(* Logix 5000 project; controller CPU_01 1756-L85E rev 36.11; software revision 36.00 *)
// CODE TESTING 20250421

TASK MainTask (continuous, watchdog 500 ms) : MainProgram, AlarmManagement, DesignPatters

MODULES
   Local : 1756-L85E (ICP 2, rev 36.11)
      INPUTS : vendor 1 type 0 code 15 (ICP 3, rev 1.1, Output RPI 50 ms)
      OUTPUT : vendor 1 type 0 code 15 (ICP 4, rev 1.1, Output RPI 50 ms)
END_MODULES

TYPE IBN_Programming :
STRUCT
   DEBUG : BOOL;   // DEBUGGING
   TODO : BOOL;   // TODO
   BYPASS : BOOL;   // BYPASS - DONOT REMOVE
   ALWAYS_OFF : BOOL;   // ALWAY OFF
   ALWAYS_ON : BOOL;   // ALWAY ON
   OUTPUTS : DINT[25];   // TEST BIT OUTPUTS
   SERIAL_NUMBER : DINT[25];   // OPEN ISSUES
END_STRUCT
END_TYPE

TYPE UDT_FiveStepMethod :
STRUCT
   TriggerPrecodition : BOOL;
   Safe : BOOL;
   Command : BOOL;
   InPosition : BOOL;
   TimeOutFault : BOOL;
END_STRUCT
END_TYPE

TYPE UDT_Missions :
STRUCT
   Missions : DINT;
   Start : DINT;
   Done : DINT;
END_STRUCT
END_TYPE

ADD_ON_INSTRUCTION AO_HANDLE_COMMAND_PANEL_BUTTONS_HARDWARE   (* revision 1.0 *)

ROUTINE Logic   (* structured text *)
   
END_ROUTINE
END_ADD_ON_INSTRUCTION

ADD_ON_INSTRUCTION AOI_Flasher   (* revision 1.0 *)
VAR_OUTPUT
   Output : BOOL; {access None, required}
END_VAR
VAR_INPUT
   TimerPreset_2 : DINT; {access None, required}
   TimerPreset_1 : DINT; {access None, required}
END_VAR
VAR
   Timer : TIMER[2]; {access None}
END_VAR

ROUTINE Logic   (* ladder *)
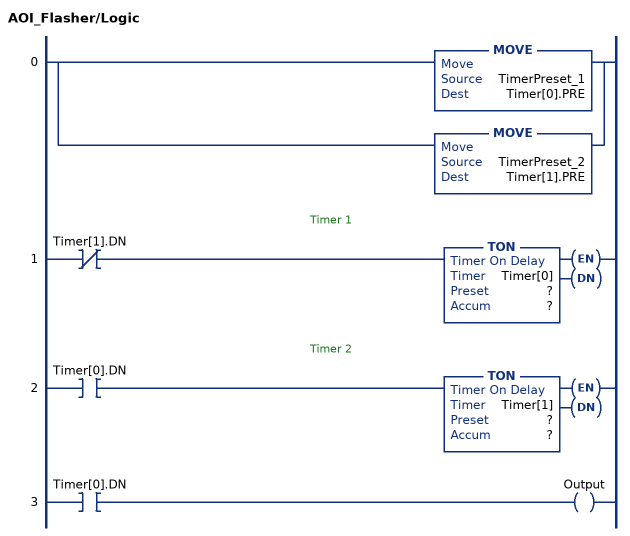
   0: [MOVE(TimerPreset_1,Timer[0].PRE) ,MOVE(TimerPreset_2,Timer[1].PRE) ];
   // Timer 1
   1: XIO(Timer[1].DN)TON(Timer[0],?,?);
   // Timer 2
   2: XIC(Timer[0].DN)TON(Timer[1],?,?);
   3: XIC(Timer[0].DN)OTE(Output);
END_ROUTINE
END_ADD_ON_INSTRUCTION

ADD_ON_INSTRUCTION AOI_Flasher_01   (* revision 1.0 *)
VAR_OUTPUT
   FLASHER_500ms_Led : BOOL; {access Read Only, required}
END_VAR
VAR
   FLASHER_500ms : FBD_TIMER; {access None}
END_VAR

ROUTINE Logic   (* structured text *)
   (* Declare Timer and Tag Variables *)
   IF NOT FLASHER_500ms.DN THEN
   	FLASHER_500ms.PRE := 1000;
   	FLASHER_500ms.EN := 1;
   	tonr(FLASHER_500ms);
   
   END_IF;
   
   IF FLASHER_500ms.ACC >= 1000 THEN
       FLASHER_500ms_Led := 1;
   ELSE
       FLASHER_500ms_Led := 0;
   END_IF;
   
   
END_ROUTINE
END_ADD_ON_INSTRUCTION

VAR_GLOBAL   (* controller tags *)
   DateTimeFromPLC : DINT[7] := ([0] := 2025, [1] := 4, [2] := 21, [3] := 16, [4] := 49, [5] := 42, [6] := 773920);
        [0]   // Year
        [1]   // Month
        [2]   // Day
        [3]   // Hours
        [4]   // Minute
        [5]   // Seconds
        [6]   // Microseconds
   IBN_DHF : IBN_Programming := (ALWAYS_ON := 1, SERIAL_NUMBER[1] := 24);
        .SERIAL_NUMBER[0].0   // 001: Timer not working
        .OUTPUTS[0].0   // 000: Spare
        .OUTPUTS[0].1   // 001: Basic Flasher bit
        .SERIAL_NUMBER[0].1   // 002: Create a trigger for getting the time
   R6 : CONTROL[25] := ([3].LEN := 4, [3].POS := 3);
   SterileWaterRinse_Array : DINT[2,20] := ([0,0] := 1, [0,1] := 2, [0,2] := 4, [0,3] := 12);
   SterileWaterRinse_Bits : DINT[8] := ([0] := 12, [2] := 7);
END_VAR

PROGRAM AlarmManagement   (* main routine R000_MainRouting *)
VAR
   AlarmMessage : BOOL[64] := ([0] := 1, [2] := 1);
        [0]   // 1000: Motor overload tripped
        [1]   // 1001: Pump over tempature
   AlarmTimers : TIMER[16] := ([0].PRE := 5000, [0].ACC := 5000, [0].EN := 1, [0].DN := 1);
   AlarmTrigger : BOOL[64];
   Messages : BOOL[64];
   MotorOverLoad : BOOL;
   MotorStart : BOOL := 1;
   PumpTemperature : DINT;
END_VAR

ROUTINE R000_MainRouting   (* structured text *)
   // Blocks
   jsr(R020_AlarmManagement);
   
END_ROUTINE

ROUTINE R020_AlarmManagement   (* ladder *)
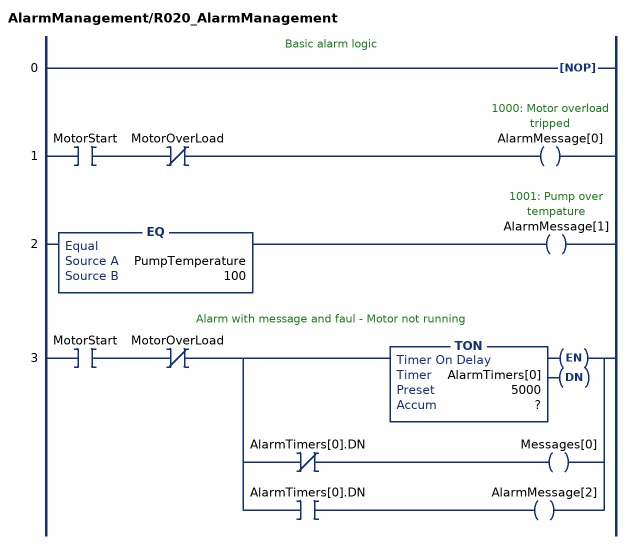
   // Basic alarm logic
   0: NOP();
   1: XIC(MotorStart)XIO(MotorOverLoad)OTE(AlarmMessage[0]);
   2: EQ(PumpTemperature,100)OTE(AlarmMessage[1]);
   // Alarm with message and faul - Motor not running
   3: XIC(MotorStart)XIO(MotorOverLoad)[TON(AlarmTimers[0],?,?) ,XIO(AlarmTimers[0].DN) OTE(Messages[0]) ,XIC(AlarmTimers[0].DN) OTE(AlarmMessage[2]) ];
END_ROUTINE
END_PROGRAM

PROGRAM DesignPatters   (* main routine R000_MainRoutine *)
VAR
   AutoMode : BOOL;
   AutoModePB : BOOL;
   Command : BOOL;
   EStopOK : BOOL;
   FaultTimeOut : BOOL;
   FaultTimer : TIMER := (PRE := 1000);
   FaultTimerReset : BOOL;
   Flasher1 : BOOL;
   Flasher_10 : AOI_Flasher_01;
   Flasher_1_sec : BOOL;
   Flasher_5000hz : AOI_Flasher := (TimerPreset_2 := 500, TimerPreset_1 := 500);
   FromSeqLogic : BOOL;
   InPosition : BOOL;
   LED : BOOL;
   LED_2 : BOOL;
   ManualMode : BOOL := 1;
   ManualModePB : BOOL;
   MissionsDone : DINT;   // Mssions complete
        .1   // Mission 1 done
   MissionsStart : DINT;   // Mssions complete
        .1   // Mission 1 done
   Mode : DINT := 1;
   ModePB : DINT := 1;
   PushButton : BOOL;
   Safe : BOOL;
   Sensor : BOOL;
   TimeOutFault : BOOL;
   TON_Flasher_1_sec : TIMER := (PRE := 2000, ACC := 147, EN := 1, TT := 1);
   TriggerPrecondition : BOOL;
   ValveMissions : UDT_Missions := (Missions := 1);
        .Missions.0   // No mission
        .Missions.1   // Mission 1
        .Missions.2   // Mission 2
END_VAR

ROUTINE R000_MainRoutine   (* ladder *)
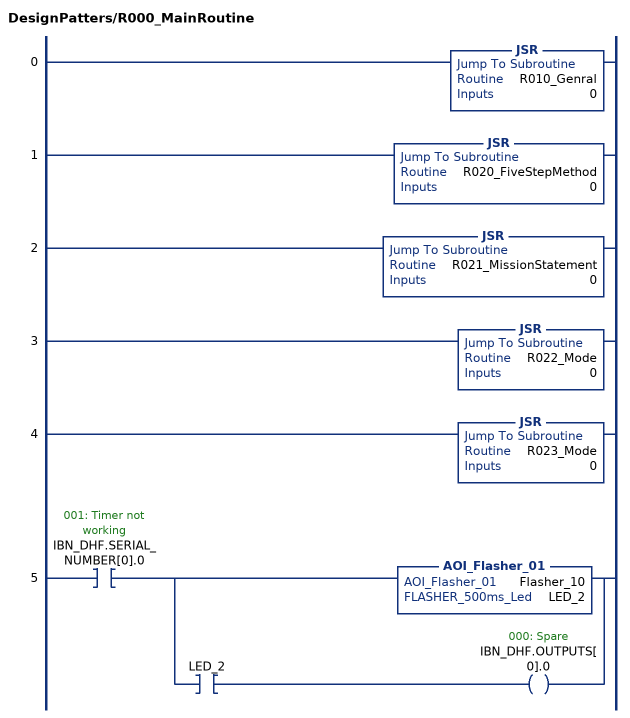
   0: JSR(R010_Genral,0);
   1: JSR(R020_FiveStepMethod,0);
   2: JSR(R021_MissionStatement,0);
   3: JSR(R022_Mode,0);
   4: JSR(R023_Mode,0);
   5: XIC(IBN_DHF.SERIAL_NUMBER[0].0)[AOI_Flasher_01(Flasher_10,LED_2) ,XIC(LED_2) OTE(IBN_DHF.OUTPUTS[0].0) ];
END_ROUTINE

ROUTINE R010_Genral   (* ladder *)
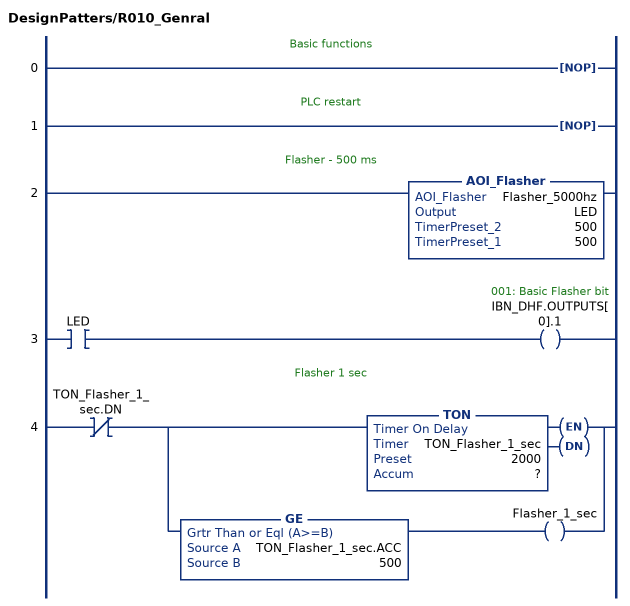
   // Basic functions
   0: NOP();
   // PLC restart
   1: NOP();
   // Flasher - 500 ms
   2: AOI_Flasher(Flasher_5000hz,LED,500,500);
   3: XIC(LED)OTE(IBN_DHF.OUTPUTS[0].1);
   // Flasher 1 sec
   4: XIO(TON_Flasher_1_sec.DN)[TON(TON_Flasher_1_sec,?,?) ,GE(TON_Flasher_1_sec.ACC,500) OTE(Flasher_1_sec) ];
END_ROUTINE

ROUTINE R020_FiveStepMethod   (* ladder *)
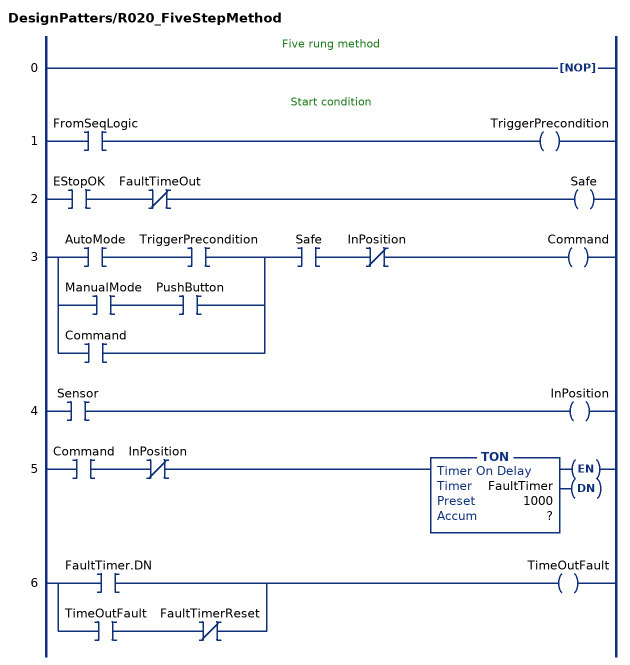
   // Five rung method
   0: NOP();
   // Start condition
   1: XIC(FromSeqLogic)OTE(TriggerPrecondition);
   2: XIC(EStopOK)XIO(FaultTimeOut)OTE(Safe);
   3: [XIC(AutoMode) XIC(TriggerPrecondition) ,XIC(ManualMode) XIC(PushButton) ,XIC(Command) ]XIC(Safe)XIO(InPosition)OTE(Command);
   4: XIC(Sensor)OTE(InPosition);
   5: XIC(Command)XIO(InPosition)TON(FaultTimer,?,?);
   6: [XIC(FaultTimer.DN) ,XIC(TimeOutFault) XIO(FaultTimerReset) ]OTE(TimeOutFault);
END_ROUTINE

ROUTINE R021_MissionStatement   (* ladder *)
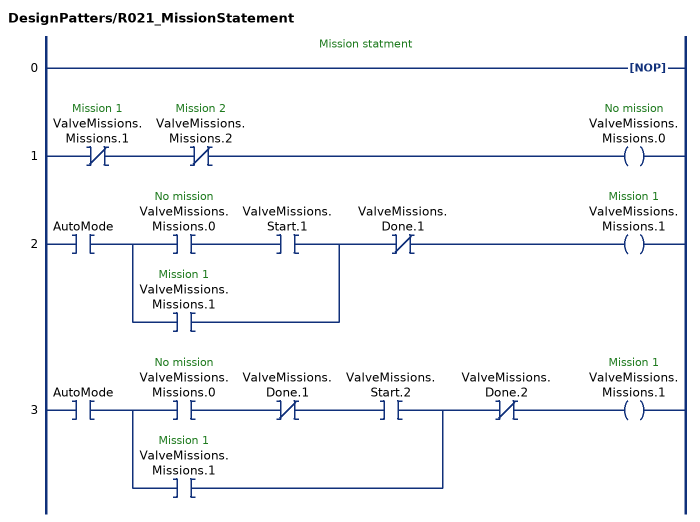
   // Mission statment
   0: NOP();
   1: XIO(ValveMissions.Missions.1)XIO(ValveMissions.Missions.2)OTE(ValveMissions.Missions.0);
   2: XIC(AutoMode)[XIC(ValveMissions.Missions.0) XIC(ValveMissions.Start.1) ,XIC(ValveMissions.Missions.1) ]XIO(ValveMissions.Done.1)OTE(ValveMissions.Missions.1);
   3: XIC(AutoMode)[XIC(ValveMissions.Missions.0) XIO(ValveMissions.Done.1) XIC(ValveMissions.Start.2) ,XIC(ValveMissions.Missions.1) ]XIO(ValveMissions.Done.2)OTE(ValveMissions.Missions.1);
END_ROUTINE

ROUTINE R022_Mode   (* ladder *)
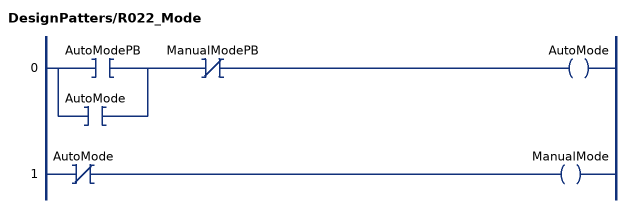
   0: [XIC(AutoModePB) ,XIC(AutoMode) ]XIO(ManualModePB)OTE(AutoMode);
   1: XIO(AutoMode)OTE(ManualMode);
END_ROUTINE

ROUTINE R023_Mode   (* ladder *)
// Three mode selection
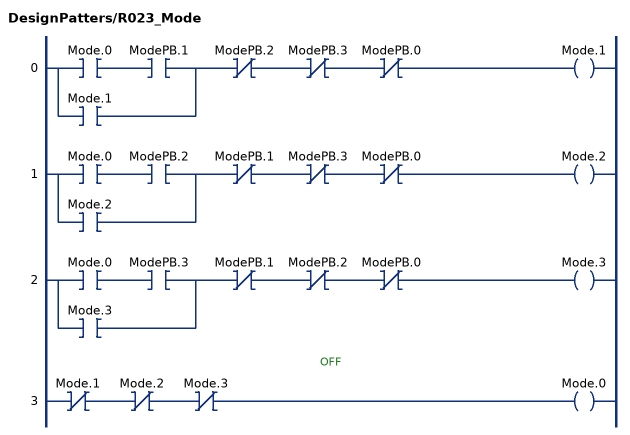
   0: [XIC(Mode.0) XIC(ModePB.1) ,XIC(Mode.1) ]XIO(ModePB.2)XIO(ModePB.3)XIO(ModePB.0)OTE(Mode.1);
   1: [XIC(Mode.0) XIC(ModePB.2) ,XIC(Mode.2) ]XIO(ModePB.1)XIO(ModePB.3)XIO(ModePB.0)OTE(Mode.2);
   2: [XIC(Mode.0) XIC(ModePB.3) ,XIC(Mode.3) ]XIO(ModePB.1)XIO(ModePB.2)XIO(ModePB.0)OTE(Mode.3);
   // OFF
   3: XIO(Mode.1)XIO(Mode.2)XIO(Mode.3)OTE(Mode.0);
END_ROUTINE
END_PROGRAM

PROGRAM MainProgram   (* main routine R000_MainRoutine *)
VAR
   FirstScan : BOOL := 1;
END_VAR

ROUTINE InformationAndHistory   (* structured text *)
   (*****************************************************************************************************************
   PROJECT:	       	Augenstein 27049 Tub Feed
   ROUTINE:			InformationAndHistory
   AUTHOR:				Esther Erickson
   CREATED:		    04.07.2007
   DESCRIPTION:		General information and revision history.
   INPUT PARAMETER:	None
   OUTPUT PARAMETER:   None
   
   *****************************************************************************************************************
   | VERSION |    DATE    |       COMMENT       | CHANGE BY |
   |---------|:----------:|:-------------------:|-----------|
   | 0.00    | 2025-04-22 |     NEW PROJECT     |           |
   | 0.01    | 2025-04-26 | Add design patterns |           |
   *****************************************************************************************************************)
   
   
   
END_ROUTINE

ROUTINE R000_MainRoutine   (* ladder *)
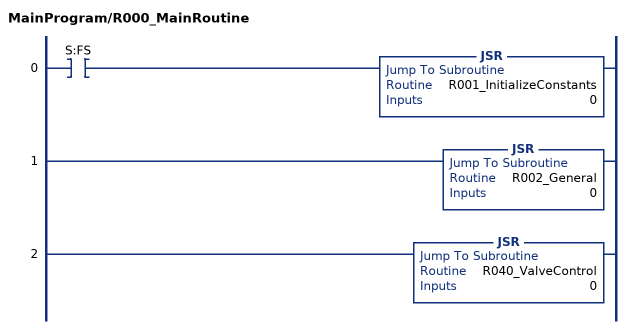
   0: XIC(S:FS)JSR(R001_InitializeConstants,0);
   1: JSR(R002_General,0);
   2: JSR(R040_ValveControl,0);
END_ROUTINE

ROUTINE R001_InitializeConstants   (* structured text *)
   // General information
   
   IBN_DHF.ALWAYS_OFF := 0;
   IBN_DHF.ALWAYS_ON := 1;
END_ROUTINE

ROUTINE R002_General   (* ladder *)
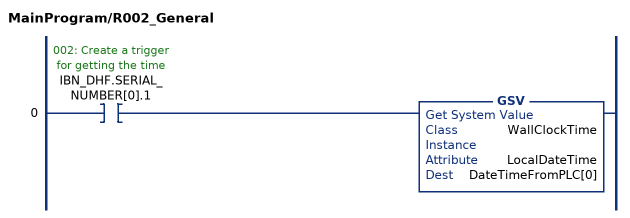
   0: XIC(IBN_DHF.SERIAL_NUMBER[0].1)GSV(WallClockTime,,LocalDateTime,DateTimeFromPLC[0]);
END_ROUTINE

ROUTINE R003_Template   (* ladder *)
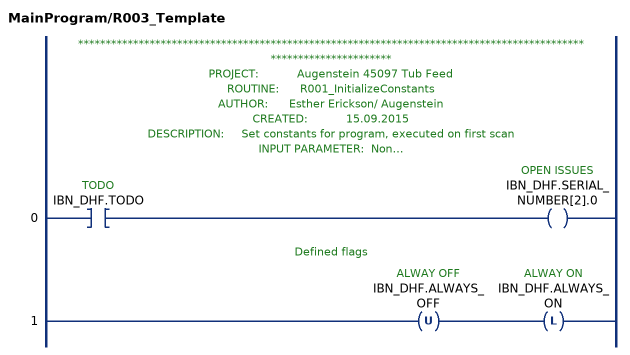
   // ******************************************************************************************************************
   // PROJECT:		       Augenstein 45097 Tub Feed
   // ROUTINE:			R001_InitializeConstants
   // AUTHOR:			Esther Erickson/ Augenstein
   // CREATED:		       15.09.2015
   // DESCRIPTION:		 Set constants for program, executed on first scan
   // INPUT PARAMETER:	None
   // OUTPUT PARAMETER:    None
   // VERSION	       DATE           COMMENT/ CHANGED BY
   // V0.00		04.07.2007		Created / EE
   // V1.00		15.09.2015		Created / EM
   // ******************************************************************************************************************
   // Used for equations that need PI as opposed to typing the number.
   0: XIC(IBN_DHF.TODO)OTE(IBN_DHF.SERIAL_NUMBER[2].0);
   // Defined flags
   1: OTU(IBN_DHF.ALWAYS_OFF)OTL(IBN_DHF.ALWAYS_ON);
END_ROUTINE

ROUTINE R040_ValveControl   (* ladder *)
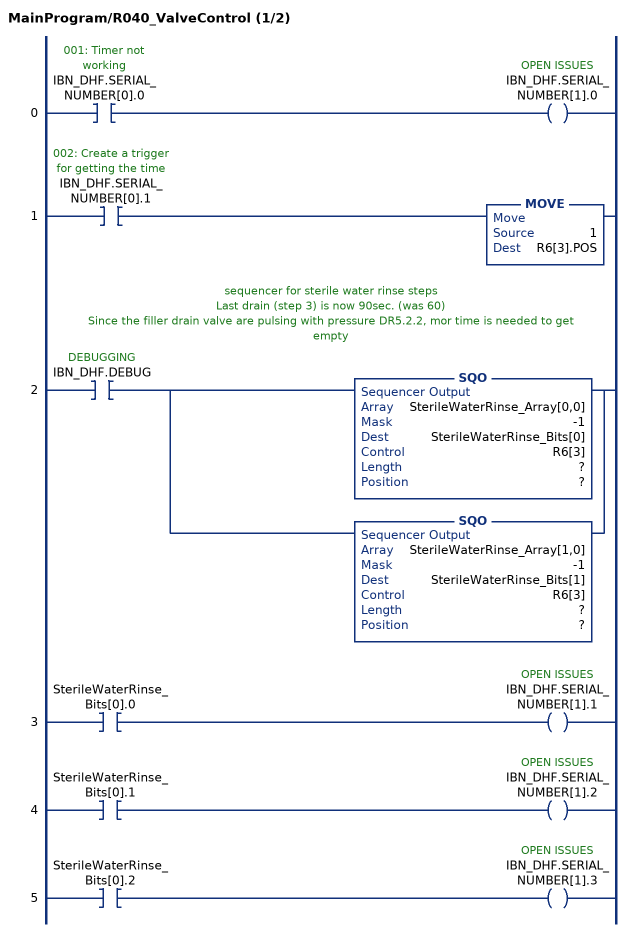
   0: XIC(IBN_DHF.SERIAL_NUMBER[0].0)OTE(IBN_DHF.SERIAL_NUMBER[1].0);
   1: XIC(IBN_DHF.SERIAL_NUMBER[0].1)MOVE(1,R6[3].POS);
   // sequencer for sterile water rinse steps
   // Last drain (step 3) is now 90sec. (was 60)
   // Since the filler drain valve are pulsing with pressure DR5.2.2, mor time is needed to get empty
   2: XIC(IBN_DHF.DEBUG)[SQO(SterileWaterRinse_Array[0,0],-1,SterileWaterRinse_Bits[0],R6[3],?,?) ,SQO(SterileWaterRinse_Array[1,0],-1,SterileWaterRinse_Bits[1],R6[3],?,?) ];
   3: XIC(SterileWaterRinse_Bits[0].0)OTE(IBN_DHF.SERIAL_NUMBER[1].1);
   4: XIC(SterileWaterRinse_Bits[0].1)OTE(IBN_DHF.SERIAL_NUMBER[1].2);
   5: XIC(SterileWaterRinse_Bits[0].2)OTE(IBN_DHF.SERIAL_NUMBER[1].3);
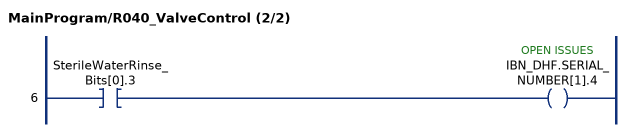
   6: XIC(SterileWaterRinse_Bits[0].3)OTE(IBN_DHF.SERIAL_NUMBER[1].4);
END_ROUTINE
END_PROGRAM
